Universal Robots PolyScope program: RC_E8_PLACE_832.urp

Program RC_E8_PLACE_832 (createdIn=3.0.0 lastSavedIn=3.0.0 directory=/programs installation=default)
Robot Program (runOnlyOnce=true motionType=MoveJ speed=1.047198 acceleration=1.396263 useActiveTCP=false)
  'Program generated by RoboDK v4.1.0 for UR3e_HORNO on 06/09/2022 17:07:23'
  'Using nominal kinematics.'
  'Using Ref. Frame Traslado C: p[0.369000, -0.220000, 0.032000, 0.000000, 0.000000, 0.000000]'
  'Using TCP 0208-0001-0001-307-000-3 Horno: p[0.000000, 0.000000, 0.164750, 0.000000, 0.000000, 0.000000]'
  Script: set_tcp(p[0.000000, 0.000000, 0.164750, 0.000000, 0.000000, 0.000000])
  Script: movej([0.420275, -1.803623, -0.993965, -3.453134, 0.446281, 0.000000],0.60000,0.12500,0,0.0000)
  MoveL speed 100 mm/s, acceleration 120 mm/s^2 (useActiveTCP=true)
    Waypoint Waypoint_1: TCP in base x=653 y=-490.005 z=179 mm, rx=1.5841 ry=-0.0094 rz=-0.0052 rad; joints [24.566, -112.37, -109.168, -136.655, 25.106, -1.486] deg; flange x=654.521 y=-325.277 z=181.204 mm, rx=1.5841 ry=-0.0094 rz=-0.0052 rad
  'Detach from 0208-0001-0001-307-000-3 Horno'
  Script: movej([0.420275, -1.803623, -0.993965, -3.453134, 0.446281, 0.000000],0.90000,0.50000,0,0.0000)
